{attribute 'obsolete' := 'Use E_MotionRequest'}
TYPE ENUM_MotionRequest : E_MotionRequest; END_TYPE

(* stored: Version 1.1.0.1
   DUT ENUM_MotionRequest: Id {0aa072d2-1d45-470d-9236-3fe22e6a4ee5} *)
